ABB RobotStudio station: TestingLetters2_20220802-123221.rsstn

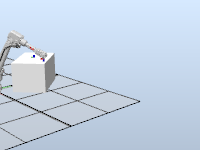
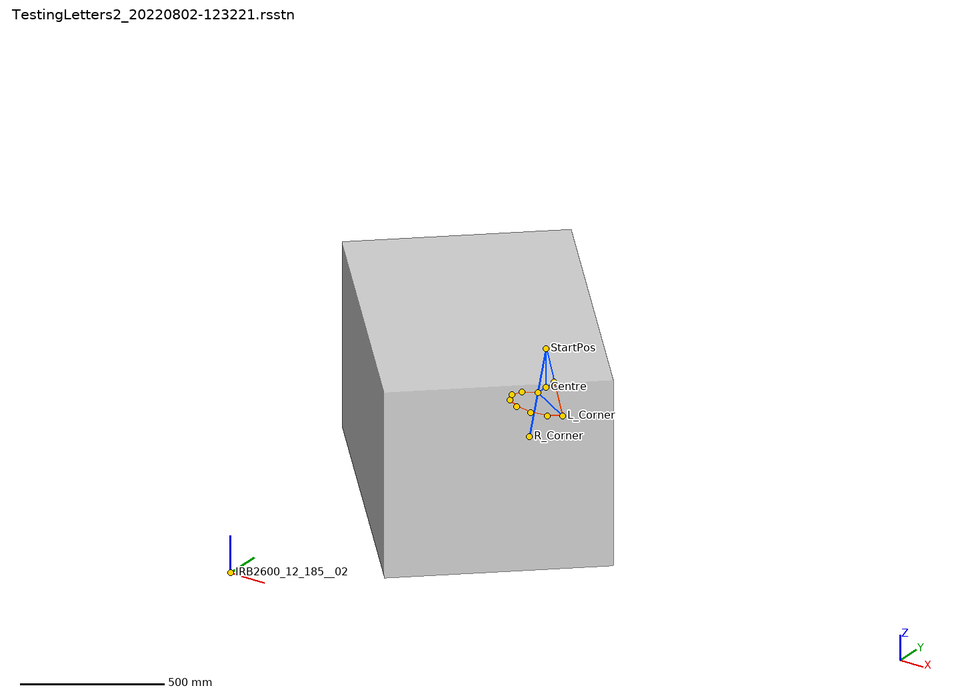
[picture v1: parts stored in the station drawn from their meshes, with robot base, taught points and paths (robot models come from the ABB library and are not in the file)]
Station TestingLetters2 (saved by RobotStudio 22.1.9826.0)
Controller IRB2600_12_185
  mechanical unit ROB_1: IRB2600_12_185__02, 6 joints, base frame (0, 0, 0) mm
Layout (positions relative to the parent item):
  - IRB2600_12_185__02 [mechanism, from Robots\IRB2600_12_185_G_02.rslib] at (0, 0, 0) mm; joint values [0.6436, 0.4918, 0.0417, 0, 1.0372, -0.1418] (rad or m)
  - Curve [part], size 204.9 x 187.3 x 188.4 mm
  - Part_1 [part], size 141.6 x 162.5 x 162.5 mm
  - BoxTable [part] at (353.59, 989.09, 715) mm, rotated rx 0 ry 0 rz 132 deg, size 1205 x 800 x 715 mm
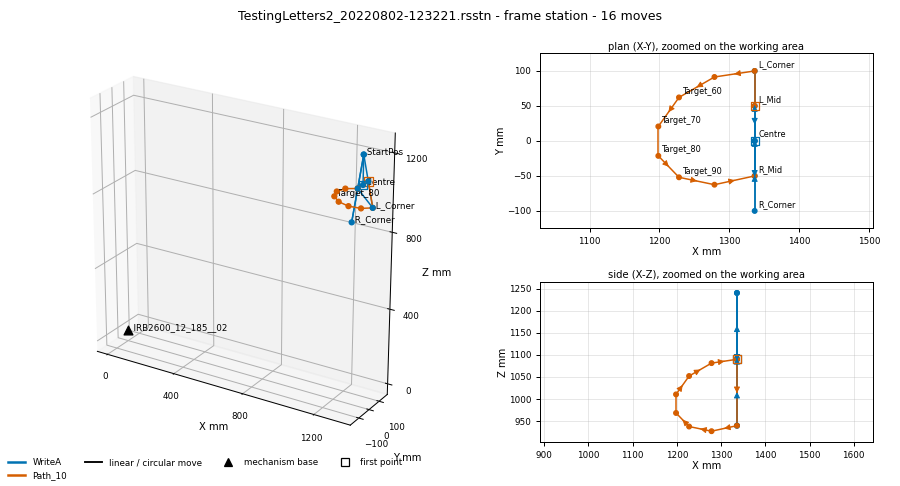
[picture p0: tool path of TestingLetters2_20220802-123221.rsstn in frame station, 16 of 16 moves have a stored position in this frame; points joined in program order, loops and branches not executed]
Targets, tools, work objects and paths stored in the station, written as RAPID:
! task T_ROB1
MODULE Module1
  CONST robtarget Centre:=[[1336.000068323,0,1090.000067718],[0.706151716,0,0.708060558,0],[0,0,0,1],[9E+09,9E+09,9E+09,9E+09,9E+09,9E+09]];
  CONST robtarget R_Corner:=[[1336.000063563,-100.000004349,940.00009488],[0.706151705,0.00000002,0.70806057,0.000000015],[-1,-1,0,1],[9E+09,9E+09,9E+09,9E+09,9E+09,9E+09]];
  CONST robtarget L_Corner:=[[1336.000063563,100.000004349,940.00009488],[0.706151705,0.000000006,0.70806057,0.000000011],[0,0,-1,1],[9E+09,9E+09,9E+09,9E+09,9E+09,9E+09]];
  CONST robtarget StartPos:=[[1336.000077935,0,1240.000023955],[0.706151706,0.000000003,0.708060568,0.000000003],[0,0,0,1],[9E+09,9E+09,9E+09,9E+09,9E+09,9E+09]];
  CONST robtarget R_Mid:=[[1336.00007495,-49.999997558,1090.000058219],[0.706151717,0,0.708060557,0.000000002],[-1,-1,0,1],[9E+09,9E+09,9E+09,9E+09,9E+09,9E+09]];
  CONST robtarget L_Mid:=[[1336.000074936,49.999998053,1090.000053177],[0.706151696,0.000000009,0.708060578,0.00000001],[0,0,-1,1],[9E+09,9E+09,9E+09,9E+09,9E+09,9E+09]];
  CONST robtarget Target_10:=[[1336,100,940],[0.999305744,-0.000691513,-0.025142572,-0.027484594],[0,1,1,2],[9E+09,9E+09,9E+09,9E+09,9E+09,9E+09]];
  CONST robtarget Target_20:=[[1194.436050583,-1.022784819,988.977215181],[0.653281482,-0.27059805,-0.27059805,-0.653281482],[0,0,0,0],[9E+09,9E+09,9E+09,9E+09,9E+09,9E+09]];
  CONST robtarget Target_30:=[[1336,-50,1090],[0.979760344,-0.00503092,0.024823562,0.198565224],[0,0,0,0],[9E+09,9E+09,9E+09,9E+09,9E+09,9E+09]];
  CONST robtarget Target_40:=[[1336.000074936,49.999998053,1090.000053177],[0.706151696,0.000000009,0.708060578,0.00000001],[0,0,-1,1],[9E+09,9E+09,9E+09,9E+09,9E+09,9E+09]];
  CONST robtarget Target_50:=[[1278.542819721,91.389446046,927.486590616],[0.999975267,0.002921695,0.000692597,-0.006360029],[0,0,0,0],[9E+09,9E+09,9E+09,9E+09,9E+09,9E+09]];
  CONST robtarget Target_60:=[[1227.863094956,62.1982137,938.045571211],[0.347421586,-0.171066931,-0.06462105,-0.919705641],[0,0,0,0],[9E+09,9E+09,9E+09,9E+09,9E+09,9E+09]];
  CONST robtarget Target_70:=[[1198.335643403,20.70611595,968.681988242],[0.543625031,-0.274973202,-0.1944354,-0.768801951],[0,0,0,0],[9E+09,9E+09,9E+09,9E+09,9E+09,9E+09]];
  CONST robtarget Target_80:=[[1198.335643403,-21.318011758,1010.70611595],[0.761374708,-0.221743362,-0.329464565,-0.51243686],[0,0,0,0],[9E+09,9E+09,9E+09,9E+09,9E+09,9E+09]];
  CONST robtarget Target_90:=[[1227.863094956,-51.954428789,1052.1982137],[0.918777516,-0.076695658,-0.317196341,-0.222153403],[0,0,0,0],[9E+09,9E+09,9E+09,9E+09,9E+09,9E+09]];
  CONST robtarget Target_100:=[[1278.542819721,-62.513409384,1081.389446046],[0.985860517,0.001511956,-0.167324226,0.008908323],[0,0,0,0],[9E+09,9E+09,9E+09,9E+09,9E+09,9E+09]];
  CONST robtarget Target_110:=[[1336,-50,1090],[0.979760344,-0.00503092,0.024823562,0.198565224],[0,0,0,0],[9E+09,9E+09,9E+09,9E+09,9E+09,9E+09]];
  PROC WriteA()
    MoveL Centre,v300,fine,tool0\WObj:=wobj0;
    MoveL StartPos,v300,fine,tool0\WObj:=wobj0;
    MoveL R_Corner,v300,fine,tool0\WObj:=wobj0;
    MoveL StartPos,v300,fine,tool0\WObj:=wobj0;
    MoveL L_Corner,v300,fine,tool0\WObj:=wobj0;
    MoveL R_Mid,v300,fine,tool0\WObj:=wobj0;
    MoveL L_Mid,v300,fine,tool0\WObj:=wobj0;
  ENDPROC
  PROC Path_10()
    MoveL Target_40,v1000,z100,tool0\WObj:=wobj0;
    MoveL Target_10,v1000,z100,tool0\WObj:=wobj0;
    MoveL Target_50,v1000,z100,tool0\WObj:=wobj0;
    MoveL Target_60,v1000,z100,tool0\WObj:=wobj0;
    MoveL Target_70,v1000,z100,tool0\WObj:=wobj0;
    MoveL Target_80,v1000,z100,tool0\WObj:=wobj0;
    MoveL Target_90,v1000,z100,tool0\WObj:=wobj0;
    MoveL Target_100,v1000,z100,tool0\WObj:=wobj0;
    MoveL Target_110,v1000,z100,tool0\WObj:=wobj0;
  ENDPROC
ENDMODULE

! task T_ROB1
MODULE CalibData
  TASK PERS wobjdata BoxTable:=[FALSE,TRUE,"",[[0,0,0],[1,0,0,0]],[[353.591,989.093,715],[0.406736643,0,0,0.913545458]]];
ENDMODULE

